FUNCTION Convert_DWORD_TO_TOD : Hresult
VAR_INPUT
	in : DWORD;
	out : REFERENCE TO TOD;
END_VAR
VAR
	converted : TOD;
END_VAR

converted := DWORD_TO_TOD(in);

IF (TOD_TO_DWORD(converted) <> in) THEN
	Convert_DWORD_TO_TOD := INCOMPATIBLE;
	RETURN;
END_IF

out := converted;

END_FUNCTION

(* stored: Version 1.1.0.1, ProductVersion 3.1.4024.12
   POU Convert_DWORD_TO_TOD: Id {ac7e15f0-7cb6-4f17-80e4-2d22db48f038}, SpecialFunc None *)
